{attribute addProperty BoxType "EK1122-0000-0018"}
{attribute addProperty Id "Beckhoff_EK18xxsub_EK1100EK1100_179A0949162A_0001_EK1814_0000_0016EK1814_E58483979612A_0002_EK1814_0000_0017EK1814_E58483979612A_0003_EK1814_0000_0018EK1814_E58483979612A_0004_EK1814_0000_0019EK1814_E58483979612A_0005_EK1818_0000_0016EK1818_BAF3593512816A_0006_EK1818_0000_0017EK1818_BAF3593512816A_0007_EK1818_0000_0018EK1818_BAF3593512816A_0008_EK1828_0000_0016EK1828_0C24FBA312816A_0009_EK1828_0000_0017EK1828_0C24FBA312816A_0010_EK1828_0000_0018EK1828_0C24FBA312816A_0011_EK1828_0010_0016EK1828_04E0E56B8811A_0012_EK1828_0010_0017EK1828_04E0E56B8811A_0013_EK1828_0010_0018EK1828_04E0E56B8811"}
{attribute addProperty CRC "3954291781"}
{attribute addProperty SizeInBites "1432"}
{attribute addProperty SizeInBytes "179"}
TYPE Beckhoff_EK18xxEK1122_EBB1B445 EXTENDS EK1122_179A0949 :
STRUCT
	{attribute addProperty Name "Beckhoff_EK18xxsub_EK1100"}
	Beckhoff_EK18xxsub_EK1100 : EK1100_179A0949;
	{attribute addProperty Name "A_0001_EK1814_0000_0016"}
	A_0001_EK1814_0000_0016 : EK1814_E5848397;
	{attribute addProperty Name "A_0002_EK1814_0000_0017"}
	A_0002_EK1814_0000_0017 : EK1814_E5848397;
	{attribute addProperty Name "A_0003_EK1814_0000_0018"}
	A_0003_EK1814_0000_0018 : EK1814_E5848397;
	{attribute addProperty Name "A_0004_EK1814_0000_0019"}
	A_0004_EK1814_0000_0019 : EK1814_E5848397;
	{attribute addProperty Name "A_0005_EK1818_0000_0016"}
	A_0005_EK1818_0000_0016 : EK1818_BAF35935;
	{attribute addProperty Name "A_0006_EK1818_0000_0017"}
	A_0006_EK1818_0000_0017 : EK1818_BAF35935;
	{attribute addProperty Name "A_0007_EK1818_0000_0018"}
	A_0007_EK1818_0000_0018 : EK1818_BAF35935;
	{attribute addProperty Name "A_0008_EK1828_0000_0016"}
	A_0008_EK1828_0000_0016 : EK1828_0C24FBA3;
	{attribute addProperty Name "A_0009_EK1828_0000_0017"}
	A_0009_EK1828_0000_0017 : EK1828_0C24FBA3;
	{attribute addProperty Name "A_0010_EK1828_0000_0018"}
	A_0010_EK1828_0000_0018 : EK1828_0C24FBA3;
	{attribute addProperty Name "A_0011_EK1828_0010_0016"}
	A_0011_EK1828_0010_0016 : EK1828_04E0E56B;
	{attribute addProperty Name "A_0012_EK1828_0010_0017"}
	A_0012_EK1828_0010_0017 : EK1828_04E0E56B;
	{attribute addProperty Name "A_0013_EK1828_0010_0018"}
	A_0013_EK1828_0010_0018 : EK1828_04E0E56B;
END_STRUCT
END_TYPE

(* stored: Version 1.2.0.0, ProductVersion 3.1.4024.9
   DUT Beckhoff_EK18xxEK1122_EBB1B445: Id {1a500cef-12f5-4fe4-adff-703446b6856c} *)
